TEXTLIST TL_E_STATION_PARAMETER_VARIANT
  0 = 'J100 V3000'
  1 = 'J100 V3500'
  2 = 'J100 V4000'
  3 = 'J200 V3000'
  4 = 'J400 V3000'
  5 = 'J120 V3500 PS0'
   = ''
END_TEXTLIST

(* stored: Version 1.1.0.1
   TextList TL_E_STATION_PARAMETER_VARIANT: Id {84cce16a-9c7b-4145-b267-a11284fcc679} *)
